TYPE MachineComSubscribe :
STRUCT
  Request : MachineComRequest; // contains booleans that are used to start a specific sequence.
  Equipment : MachineComSubscribeEquipment;  // structs for equipment objects which are used by the bridges
END_STRUCT
END_TYPE

(* stored: Version 1.1.0.1
   DUT MachineComSubscribe: Id {49516409-eedf-4113-9331-838875845511} *)
